RoboDK station: ini_pos.rdk

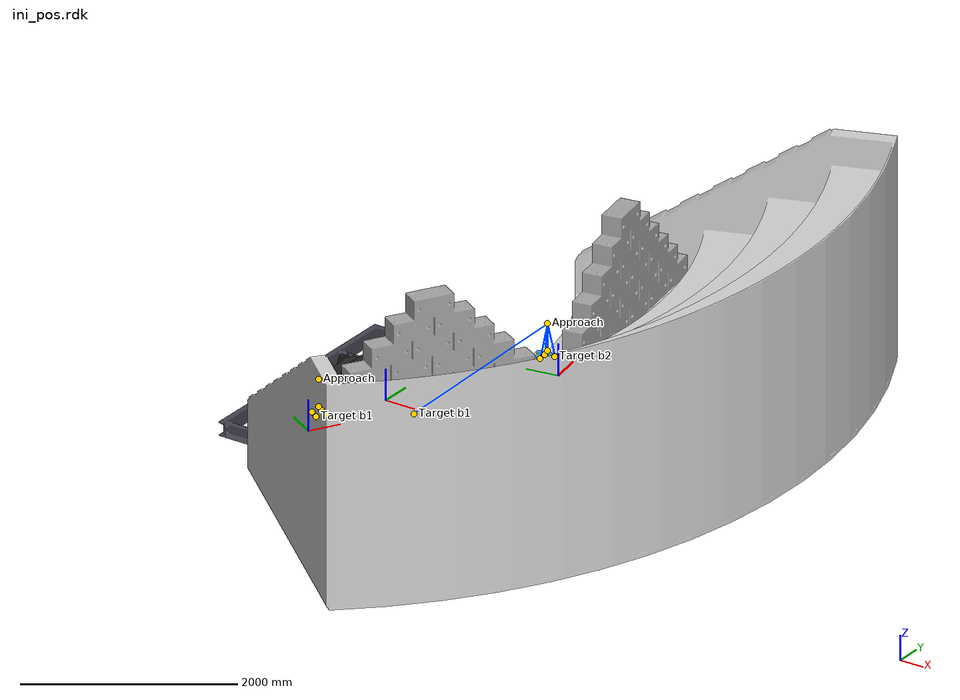
[picture v0: the station drawn from its stored meshes, robots at their saved joint values, targets as dots, program paths as lines]
Station ini_pos (saved by RoboDK 5.4.1). Poses are relative to the parent item; angles as X-Y-Z fixed-axis rotations.
  - frame KUKA KR 210-2 Base at (0, 0, 0) mm
    - robot KUKA KR 210-2: 6 axes, payload 210 kg, reach 2700 mm, repeatability 0.06 mm, weight 1267 kg
        joint limits [-185, -146, -119, -350, -125, -350] to [185, 0, 155, 350, 125, 350]; home [0, -90, 90, 0, 0, 0]; saved at [58.346, -82.845, 89.745, 86.305, -58.537, -82.19]
      - tool NEMO_TOOL, TCP at (0, 0, 200) mm, size 500 x 350 x 427.5 mm
    - object Stairs_v1 at (-2520, 0, 0) mm, size 7409.2 x 2302 x 3902.7 mm, geometry from Stairs_v1.3ds
    - frame Table 1 at (1940, -11.06, 800) mm, rotated rx 0 ry 0 rz 100 deg
      - target Approach (Cartesian target) at (200, 200, 400) mm, rotated rx -180 ry 0 rz -180 deg; joints [-42.973, 13.47, -8.834, -85.041, -43.174, 83.215] of KUKA KR 210-2
      - target Target b1 (Cartesian target) at (-272.12, 1336.14, -547.04) mm, rotated rx 180 ry 89.53 rz 80 deg; joints [26.923, -51.043, 119.863, 28.659, -70.748, -9.979] of KUKA KR 210-2
      - target Target b2 (Cartesian target) at (250, 150, 50) mm, rotated rx -180 ry 0 rz 180 deg; joints [-43.119, 28.404, 5.363, 120.692, 52.642, -134.368] of KUKA KR 210-2
      - target Target b3 (Cartesian target) at (150, 250, 50) mm, rotated rx -180 ry 0 rz 180 deg; joints [-42.803, 18.858, 20.461, 124.38, 55.416, -140.321] of KUKA KR 210-2
      - target Target b4 (Cartesian target) at (250, 250, 50) mm, rotated rx -180 ry 0 rz 180 deg; joints [-38.55, 23.97, 12.589, 126.778, 51.084, -139.956] of KUKA KR 210-2
      - target Target b5 (Cartesian target) at (200, 200, 120.71) mm, rotated rx -180 ry 0 rz 180 deg; joints [-42.973, 109.891, -190.02, 43.4, 82.794, -6.764] of KUKA KR 210-2
      - object base at (0, 0, 0) mm, size 400 x 400 x 34.3 mm
      - object row5brick1 at (1070, 0, 1000) mm, size 400 x 200 x 210 mm, geometry from brick.stp
      - object row5brick1 at (860, 0, 800) mm, size 400 x 200 x 210 mm, geometry from brick.stp
        - object brick4 at (420, 0, 0) mm, size 400 x 200 x 210 mm, geometry from brick.stp
      - object row4brick1 at (640, 0, 600) mm, size 400 x 200 x 210 mm, geometry from brick.stp
        - object brick4 at (420, 0, 0) mm, size 400 x 200 x 210 mm, geometry from brick.stp
          - object brick4 at (420, 0, 0) mm, size 400 x 200 x 210 mm, geometry from brick.stp
      - object row3brick1 at (420, 0, 400) mm, size 400 x 200 x 210 mm, geometry from brick.stp
        - object brick4 at (420, 0, 0) mm, size 400 x 200 x 210 mm, geometry from brick.stp
          - object brick4 at (420, 0, 0) mm, size 400 x 200 x 210 mm, geometry from brick.stp
            - object brick4 at (420, 0, 0) mm, size 400 x 200 x 210 mm, geometry from brick.stp
      - object row1brick1 at (0, 0, 0) mm, size 400 x 200 x 210 mm, geometry from brick.stp
        - object row1brick2 at (420, 0, 0) mm, size 400 x 200 x 210 mm, geometry from brick.stp
          - object brick1 at (420, 0, 0) mm, size 400 x 200 x 210 mm, geometry from brick.stp
            - object brick1 at (420, 0, 0) mm, size 400 x 200 x 210 mm, geometry from brick.stp
              - object brick1 at (420, 0, 0) mm, size 400 x 200 x 210 mm, geometry from brick.stp
                - object brick1 at (420, 0, 0) mm, size 400 x 200 x 210 mm, geometry from brick.stp
      - object row2brick1 at (210, 0, 200) mm, size 400 x 200 x 210 mm, geometry from brick.stp
        - object brick4 at (420, 0, 0) mm, size 400 x 200 x 210 mm, geometry from brick.stp
          - object brick4 at (420, 0, 0) mm, size 400 x 200 x 210 mm, geometry from brick.stp
            - object brick4 at (420, 0, 0) mm, size 400 x 200 x 210 mm, geometry from brick.stp
              - object brick4 at (420, 0, 0) mm, size 400 x 200 x 210 mm, geometry from brick.stp
    - object Frame at (0, 0, 0) mm, size 2000 x 2500 x 199.8 mm, geometry from Frame.stp
    - frame Table 2 at (730, -2281.06, 800) mm, rotated rx 0 ry 0 rz 60 deg
      - target Approach (Cartesian target) at (200, 200, 400) mm, rotated rx -180 ry 0 rz -180 deg; joints [-42.973, 13.47, -8.834, -85.041, -43.174, 83.215] of KUKA KR 210-2
      - target Target b1 (Cartesian target) at (150, 150, 50) mm, rotated rx -180 ry 0 rz -180 deg; joints [-47.421, 23.634, 13.122, -61.195, -57.174, 44.592] of KUKA KR 210-2
      - target Target b2 (Cartesian target) at (250, 150, 50) mm, rotated rx -180 ry 0 rz 180 deg; joints [-43.119, 28.404, 5.363, 120.692, 52.642, -134.368] of KUKA KR 210-2
      - target Target b3 (Cartesian target) at (150, 250, 50) mm, rotated rx -180 ry 0 rz 180 deg; joints [-42.803, 18.858, 20.461, 124.38, 55.416, -140.321] of KUKA KR 210-2
      - target Target b4 (Cartesian target) at (250, 250, 50) mm, rotated rx -180 ry 0 rz 180 deg; joints [-38.55, 23.97, 12.589, 126.778, 51.084, -139.956] of KUKA KR 210-2
      - target Target b5 (Cartesian target) at (200, 200, 120.71) mm, rotated rx -180 ry 0 rz 180 deg; joints [-42.973, 109.891, -190.02, 43.4, 82.794, -6.764] of KUKA KR 210-2
      - object base at (0, 0, 0) mm, size 400 x 400 x 34.3 mm
      - object row5brick1 at (1070, 0, 1000) mm, size 400 x 200 x 210 mm, geometry from brick.stp
      - object row5brick1 at (860, 0, 800) mm, size 400 x 200 x 210 mm, geometry from brick.stp
        - object brick4 at (420, 0, 0) mm, size 400 x 200 x 210 mm, geometry from brick.stp
      - object row4brick1 at (640, 0, 600) mm, size 400 x 200 x 210 mm, geometry from brick.stp
        - object brick4 at (420, 0, 0) mm, size 400 x 200 x 210 mm, geometry from brick.stp
          - object brick4 at (420, 0, 0) mm, size 400 x 200 x 210 mm, geometry from brick.stp
      - object row3brick1 at (420, 0, 400) mm, size 400 x 200 x 210 mm, geometry from brick.stp
        - object brick4 at (420, 0, 0) mm, size 400 x 200 x 210 mm, geometry from brick.stp
          - object brick4 at (420, 0, 0) mm, size 400 x 200 x 210 mm, geometry from brick.stp
            - object brick4 at (420, 0, 0) mm, size 400 x 200 x 210 mm, geometry from brick.stp
      - object row1brick1 at (0, 0, 0) mm, size 400 x 200 x 210 mm, geometry from brick.stp
        - object row1brick2 at (420, 0, 0) mm, size 400 x 200 x 210 mm, geometry from brick.stp
          - object brick1 at (420, 0, 0) mm, size 400 x 200 x 210 mm, geometry from brick.stp
            - object brick1 at (420, 0, 0) mm, size 400 x 200 x 210 mm, geometry from brick.stp
              - object brick1 at (420, 0, 0) mm, size 400 x 200 x 210 mm, geometry from brick.stp
                - object brick1 at (420, 0, 0) mm, size 400 x 200 x 210 mm, geometry from brick.stp
      - object row2brick1 at (210, 0, 200) mm, size 400 x 200 x 210 mm, geometry from brick.stp
        - object brick4 at (420, 0, 0) mm, size 400 x 200 x 210 mm, geometry from brick.stp
          - object brick4 at (420, 0, 0) mm, size 400 x 200 x 210 mm, geometry from brick.stp
            - object brick4 at (420, 0, 0) mm, size 400 x 200 x 210 mm, geometry from brick.stp
              - object brick4 at (420, 0, 0) mm, size 400 x 200 x 210 mm, geometry from brick.stp
  - program Pick and place (63 instructions, listed below)
  - program Replace objects (1 instructions, listed below)
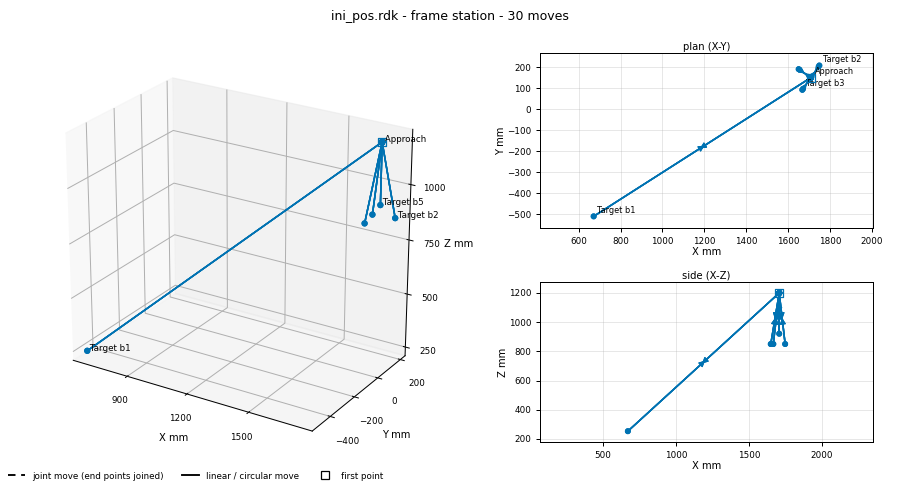
[picture p0: tool path of ini_pos.rdk in frame station, 30 of 30 moves have a stored position in this frame; points joined in program order, loops and branches not executed]

--- program Pick and place (robot KUKA KR 210-2) ---
  Set Frame: Table 1
  Set Tool: Tool at (125, 0, 100) mm, rotated rx 0 ry 90 rz 0 deg
  MoveJ (Approach)
  MoveL (Target b5)
  Attach to Tool
  Call AirValve_On
  MoveL (Approach)
  Set Frame: Table 2 at (1500, 630.03, 534.2) mm
  MoveJ (Approach)
  MoveL (Target b1)
  Detach from Tool
  Call AirValve_Off
  MoveL (Approach)
  Set Frame: Table 1
  MoveJ (Approach)
  MoveL (Target b4)
  Attach to Tool
  Call AirValve_On
  MoveL (Approach)
  Set Frame: Table 2 at (1500, 630.03, 534.2) mm
  MoveJ (Approach)
  MoveL (Target b2)
  Detach from Tool
  Call AirValve_Off
  MoveL (Approach)
  Set Frame: Table 1
  MoveJ (Approach)
  MoveL (Target b3)
  Attach to Tool
  Call AirValve_On
  MoveL (Approach)
  Set Frame: Table 2 at (1500, 630.03, 534.2) mm
  MoveJ (Approach)
  MoveL (Target b3)
  Detach from Tool
  Call AirValve_Off
  MoveL (Approach)
  Set Frame: Table 1
  MoveJ (Approach)
  MoveL (Target b2)
  Attach to Tool
  Call AirValve_On
  MoveL (Approach)
  Set Frame: Table 2 at (1500, 630.03, 534.2) mm
  MoveJ (Approach)
  MoveL (Target b4)
  Detach from Tool
  Call AirValve_Off
  MoveL (Approach)
  Set Frame: Table 1
  MoveJ (Approach)
  MoveL (Target b1)
  Attach to Tool
  Call AirValve_On
  MoveL (Approach)
  Set Frame: Delivery table at (1500, 630.03, 534.2) mm
  MoveJ (Approach)
  MoveL (Target b5)
  Detach from Tool
  Call AirValve_Off
  MoveL (Approach)
  Pause 5000 ms
  Call Replace objects

--- program Replace objects (robot KUKA KR 210-2) ---
  Replace objects
